FUNCTION_BLOCK Q_SelectColourMap (* Command Select Colour Map ( VT version 4 and later ) ( Part 6 - F.60 ) *)
  (* Standard: ISO 11783-6; Description: The Select Colour Map command is used to select the active Colour Map. This command can take a long time to execute. The command applies to any presentation from the originating Working Set, which includes objects that may be shown on other Working Set screens (e.g. Auxiliary Control objects as may be presented on VT proprietary and other Working Set masks using the Auxiliary Control Designator Type 2 Object Pointer). Return values iso_s16 - E_NO_ERR - OK - E_OVERFLOW - buffer overflow - E_NOACT - Command not possible in current state - E_NO_INSTANCE - No VT client available *)
  (* Version 1.0, 2022-07-08, franz *)
  (* Documentation:
  The Select Colour Map command is used to select the active Colour Map. This command can take a long time to execute. The command applies to any presentation from the originating Working Set, which includes objects that may be shown on other Working Set screens (e.g. Auxiliary Control objects as may be presented on VT proprietary and other Working Set masks using the Auxiliary Control Designator Type 2 Object Pointer).
   Return values
   iso_s16
    - E_NO_ERR - OK
   - E_OVERFLOW - buffer overflow
   - E_NOACT - Command not possible in current state
   - E_NO_INSTANCE - No VT client available
  *)
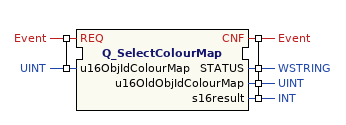
  EVENT_INPUT
    REQ WITH u16ObjIdColourMap; (* Service Request *)
  END_EVENT
  EVENT_OUTPUT
    CNF WITH STATUS, s16result, u16OldObjIdColourMap; (* Confirmation of Requested Service *)
  END_EVENT
  VAR_INPUT
    u16ObjIdColourMap : UINT; (* Object ID of Colour map object or FFFF to restore the default colour table (see A.3) *)
  END_VAR
  VAR_OUTPUT
    STATUS : WSTRING; (* Service Status *)
    u16OldObjIdColourMap : UINT; (* Old object ID of Colour map object or FFFF to restore the default colour table (see A.3) *)
    s16result : INT; (* retval see description *)
  END_VAR
END_FUNCTION_BLOCK
